(* Logix 5000 project; controller ODSI_Testing vendor 1 type 14 code 151 rev 20.19; software revision 20.05 *)

TASK MainTask (continuous, watchdog 500 ms) : MainProgram

MODULES
   Local : vendor 1 type 14 code 151 (Compact 0, rev 20.19)
      ExpansionInput : 1769-IQ16 (Compact 4, rev 1.1, Input RPI 20 ms)   // Sink or Source
      Discrete_IO : Embedded (Compact 1, rev 3.1, Output RPI 20 ms)
      Analog_IO : Embedded (Compact 2, rev 1.1, Output RPI 80 ms)
      Counters : Embedded (Compact 3, rev 1.1, Output RPI 20 ms)
END_MODULES

VAR_GLOBAL   (* controller tags *)
   DutyCycleOutput : BOOL := 1;   // 1.25 second duty cycle output
   DutyCycleTimer : TIMER := (PRE := 2500, ACC := 2111, EN := 1, TT := 1);   // Accumulates preset time then resets
   HMI_Stop_R1 : BOOL;   // Stop PB on HMI
   HMI_Stop_R2 : BOOL;   // Stop PB on HMI
   ODSI_Fail_Sample1_R1 : ALIAS FOR Local:4:I.Data.4;   // ODSI sent a fail signal for sample 1
   ODSI_Fail_Sample1_R2 : ALIAS FOR Local:1:I.Data.4;   // ODSI sent a fail signal for sample 1
   ODSI_Fail_Sample2_R1 : ALIAS FOR Local:4:I.Data.6;   // ODSI sent a fail signal for sample 2
   ODSI_Fail_Sample2_R2 : ALIAS FOR Local:1:I.Data.6;   // ODSI sent a fail signal for sample 2
   ODSI_Fail_Sample3_R1 : ALIAS FOR Local:4:I.Data.8;   // ODSI sent a fail signal for sample 3
   ODSI_Fail_Sample3_R2 : ALIAS FOR Local:1:I.Data.8;   // ODSI sent a fail signal for sample 3
   ODSI_Pass_Sample1_R1 : ALIAS FOR Local:4:I.Data.3;   // ODSI sent a pass signal for sample 1
   ODSI_Pass_Sample1_R2 : ALIAS FOR Local:1:I.Data.3;   // ODSI sent a pass signal for sample 1
   ODSI_Pass_Sample2_R1 : ALIAS FOR Local:4:I.Data.5;   // ODSI sent a pass signal for sample 2
   ODSI_Pass_Sample2_R2 : ALIAS FOR Local:1:I.Data.5;   // ODSI sent a pass signal for sample 2
   ODSI_Pass_Sample3_R1 : ALIAS FOR Local:4:I.Data.7;   // ODSI sent a pass signal for sample 3
   ODSI_Pass_Sample3_R2 : ALIAS FOR Local:1:I.Data.7;   // ODSI sent a pass signal for sample 3
   ODSI_Valve1_R1 : ALIAS FOR Local:4:I.Data.0;   // ODSI requests to open valve 1
   ODSI_Valve1_R2 : ALIAS FOR Local:1:I.Data.0;   // ODSI requests to open valve 1
   ODSI_Valve2_R1 : ALIAS FOR Local:4:I.Data.1;   // ODSI requests to open valve 2
   ODSI_Valve2_R2 : ALIAS FOR Local:1:I.Data.1;   // ODSI requests to open valve 2
   ODSI_Valve3_R1 : ALIAS FOR Local:4:I.Data.2;   // ODSI requests to open valve 3
   ODSI_Valve3_R2 : ALIAS FOR Local:1:I.Data.2;   // ODSI requests to open valve 3
   R1_DELAY_ONS : BOOL;
   R2_DELAY_ONS : BOOL;
   RandomDelay : DINT := 11;   // Random number generator 0-19
   RandomDelayDisplay_R1 : DINT;   // Snapshot of random delay at time of valve position request for remote 1
   RandomDelayDisplay_R2 : DINT;   // Snapshot of random delay at time of valve position request for remote 2
   RNG_Delay_Active_R1 : BOOL;   // HMI PB randomizing valve open delay
   RNG_Delay_Active_R2 : BOOL;   // HMI PB randomizing valve open delay
   S1_PB_Input_R1 : BOOL;   // HMI PB requesting sample 1
   S1_PB_Input_R2 : BOOL;   // HMI PB requesting sample 1
   S1_Request_R1 : ALIAS FOR Local:1:O.Data.8;   // Output to ODSI to request Sample 1
   S1_Request_R2 : ALIAS FOR Local:1:O.Data.0;   // Output to ODSI to request Sample 1
   S2_PB_Input_R1 : BOOL;   // HMI PB requesting sample 2
   S2_PB_Input_R2 : BOOL;   // HMI PB requesting sample 2
   S2_Request_R1 : ALIAS FOR Local:1:O.Data.9;   // Output to ODSI to request Sample 2
   S2_Request_R2 : ALIAS FOR Local:1:O.Data.1;   // Output to ODSI to request Sample 2
   S3_PB_Input_R1 : BOOL;   // HMI PB requesting sample 3
   S3_PB_Input_R2 : BOOL;   // HMI PB requesting sample 3
   S3_Request_R1 : ALIAS FOR Local:1:O.Data.10;   // Output to ODSI to request Sample 3
   S3_Request_R2 : ALIAS FOR Local:1:O.Data.2;   // Output to ODSI to request Sample 3
   System_Running_Display_R1 : BOOL;   // Displays system running on HMI
   System_Running_Display_R2 : BOOL;   // Displays system running on HMI
   System_Running_R1 : ALIAS FOR Local:4:I.Data.9;   // ODSI signal that indicates the system is currently analyzing a sample
   System_Running_R2 : ALIAS FOR Local:1:I.Data.9;   // ODSI signal that indicates the system is currently analyzing a sample
   SystemTime : DINT[7] := ([0] := 1998, [1] := 1, [2] := 22, [3] := 5, [4] := 42, [5] := 32, [6] := 563285);
        [1]   // Month
        [4]   // Minute
        [0]   // Year
        [2]   // Day
        [3]   // Hour
        [5]   // Second
        [6]   // Microsecond
   Temp : DINT := 10;
   Valve1_Open_Delay_R1 : TIMER;   // Delay after Request is Initiated from ODSI
   Valve1_Open_Delay_R2 : TIMER;   // Delay after Request is Initiated from ODSI
   Valve1_Open_R1 : ALIAS FOR Local:1:O.Data.11;   // Output to ODSI confirming valve 1 is open
   Valve1_Open_R2 : ALIAS FOR Local:1:O.Data.3;   // Output to ODSI confirming valve 1 is open
   Valve1_Open_Random_Delay_R1 : TIMER := (PRE := 11000);   // Randomized delay after request for valve position is received from ODSI
   Valve1_Open_Random_Delay_R2 : TIMER := (PRE := 11000);   // Randomized delay after request for valve position is received from ODSI
   Valve2_Open_Delay_R1 : TIMER;   // Delay after Request is Initiated from ODSI
   Valve2_Open_Delay_R2 : TIMER;   // Delay after Request is Initiated from ODSI
   Valve2_Open_R1 : ALIAS FOR Local:1:O.Data.12;   // Output to ODSI confirming valve 2 is open
   Valve2_Open_R2 : ALIAS FOR Local:1:O.Data.4;   // Output to ODSI confirming valve 2 is open
   Valve2_Open_Random_Delay_R1 : TIMER := (PRE := 11000);   // Randomized delay after request for valve position is received from ODSI
   Valve2_Open_Random_Delay_R2 : TIMER := (PRE := 11000);   // Randomized delay after request for valve position is received from ODSI
   Valve3_Open_Delay_R1 : TIMER;   // Delay after Request is Initiated from ODSI
   Valve3_Open_Delay_R2 : TIMER;   // Delay after Request is Initiated from ODSI
   Valve3_Open_R1 : ALIAS FOR Local:1:O.Data.13;   // Output to ODSI confirming valve 3 is open
   Valve3_Open_R2 : ALIAS FOR Local:1:O.Data.5;   // Output to ODSI confirming valve 3 is open
   Valve3_Open_Random_Delay_R1 : TIMER := (PRE := 11000);   // Randomized delay after request for valve position is received from ODSI
   Valve3_Open_Random_Delay_R2 : TIMER := (PRE := 11000);   // Randomized delay after request for valve position is received from ODSI
   Valve_Block_R1 : BOOL;   // HMI PB to prevent valves from opening
   Valve_Block_R2 : BOOL;   // HMI PB to prevent valves from opening
   Valve_Delay_R1 : DINT;
   Valve_Delay_R2 : DINT;
   Valve_Open_Delay_R2 : TIMER := (PRE := 10000);   // Delay after Request is Initiated from ODSI
END_VAR

PROGRAM MainProgram   (* main routine MainRoutine *)

ROUTINE MainRoutine   (* ladder *)
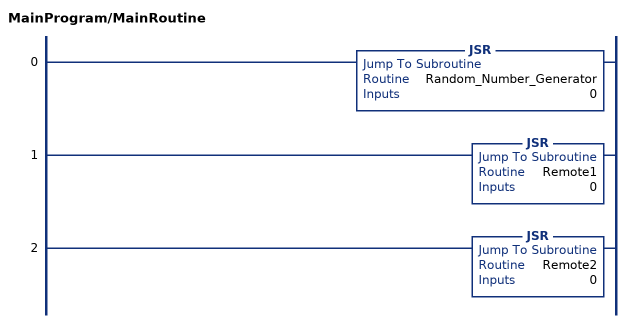
   0: JSR(Random_Number_Generator,0);
   1: JSR(Remote1,0);
   2: JSR(Remote2,0);
END_ROUTINE

ROUTINE Random_Number_Generator   (* ladder *)
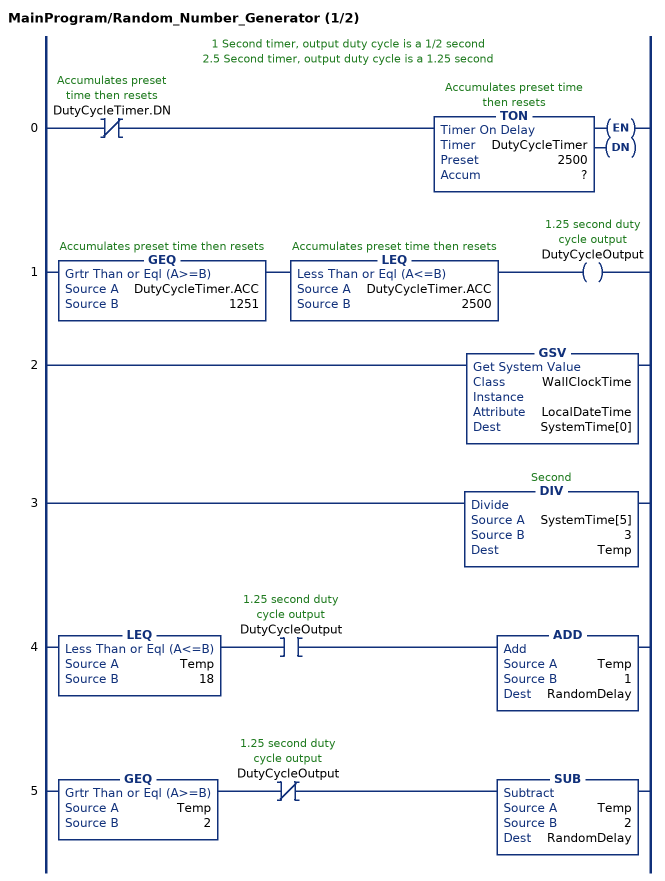
   // 1 Second timer, output duty cycle is a 1/2 second
   // 2.5 Second timer, output duty cycle is a 1.25 second
   0: XIO(DutyCycleTimer.DN)TON(DutyCycleTimer,?,?);
   1: GEQ(DutyCycleTimer.ACC,1251)LEQ(DutyCycleTimer.ACC,2500)OTE(DutyCycleOutput);
   2: GSV(WallClockTime,,LocalDateTime,SystemTime[0]);
   3: DIV(SystemTime[5],3,Temp);
   4: LEQ(Temp,18)XIC(DutyCycleOutput)ADD(Temp,1,RandomDelay);
   5: GEQ(Temp,2)XIO(DutyCycleOutput)SUB(Temp,2,RandomDelay);
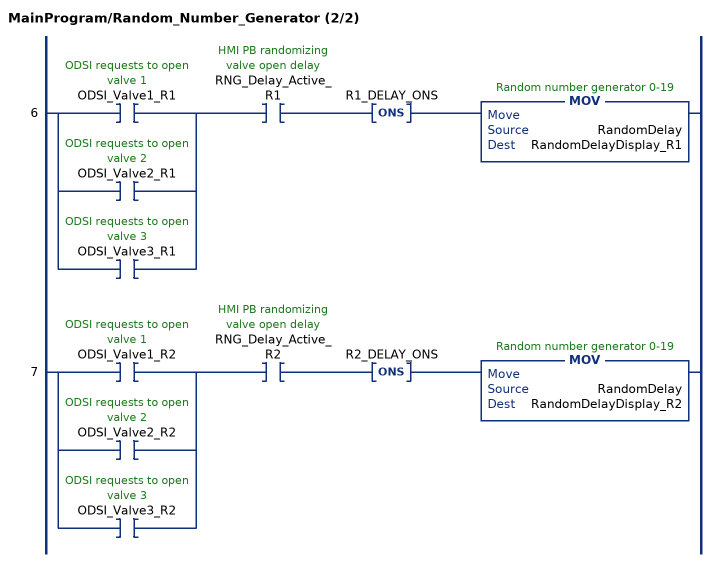
   6: [XIC(ODSI_Valve1_R1) ,XIC(ODSI_Valve2_R1) ,XIC(ODSI_Valve3_R1) ]XIC(RNG_Delay_Active_R1)ONS(R1_DELAY_ONS)MOV(RandomDelay,RandomDelayDisplay_R1);
   7: [XIC(ODSI_Valve1_R2) ,XIC(ODSI_Valve2_R2) ,XIC(ODSI_Valve3_R2) ]XIC(RNG_Delay_Active_R2)ONS(R2_DELAY_ONS)MOV(RandomDelay,RandomDelayDisplay_R2);
END_ROUTINE

ROUTINE Remote1   (* ladder *)
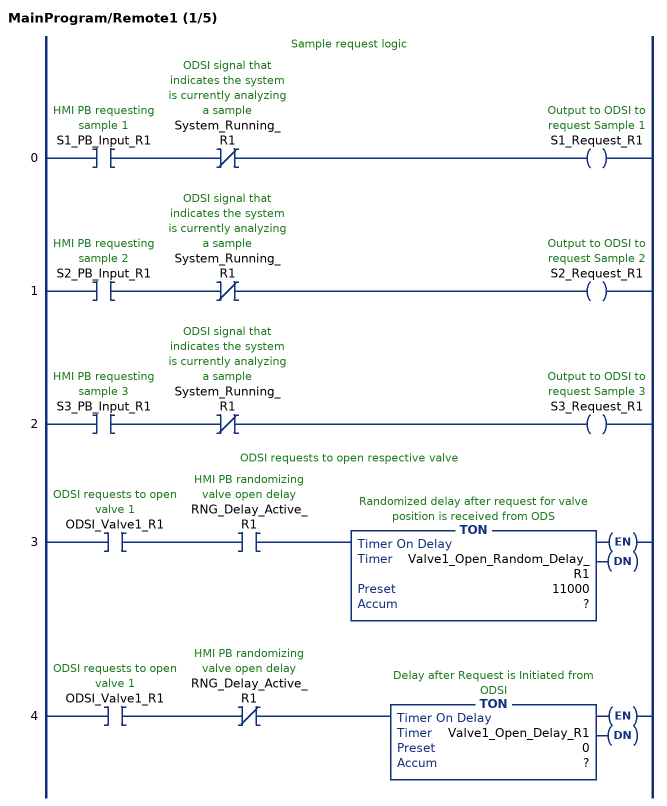
   // Sample request logic
   0: XIC(S1_PB_Input_R1)XIO(System_Running_R1)OTE(S1_Request_R1);
   1: XIC(S2_PB_Input_R1)XIO(System_Running_R1)OTE(S2_Request_R1);
   2: XIC(S3_PB_Input_R1)XIO(System_Running_R1)OTE(S3_Request_R1);
   // ODSI requests to open respective valve
   3: XIC(ODSI_Valve1_R1)XIC(RNG_Delay_Active_R1)TON(Valve1_Open_Random_Delay_R1,?,?);
   4: XIC(ODSI_Valve1_R1)XIO(RNG_Delay_Active_R1)TON(Valve1_Open_Delay_R1,?,?);
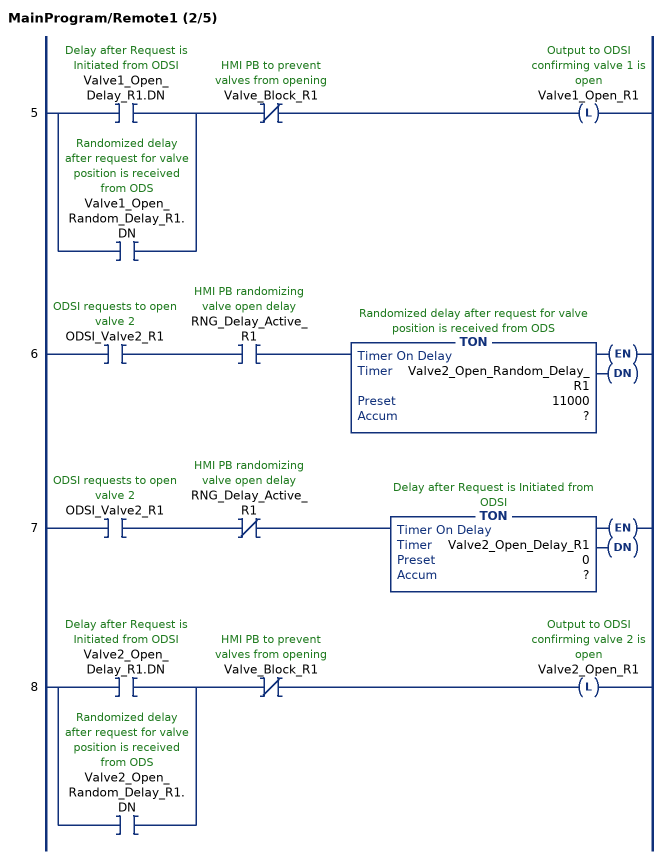
   5: [XIC(Valve1_Open_Delay_R1.DN) ,XIC(Valve1_Open_Random_Delay_R1.DN) ]XIO(Valve_Block_R1)OTL(Valve1_Open_R1);
   6: XIC(ODSI_Valve2_R1)XIC(RNG_Delay_Active_R1)TON(Valve2_Open_Random_Delay_R1,?,?);
   7: XIC(ODSI_Valve2_R1)XIO(RNG_Delay_Active_R1)TON(Valve2_Open_Delay_R1,?,?);
   8: [XIC(Valve2_Open_Delay_R1.DN) ,XIC(Valve2_Open_Random_Delay_R1.DN) ]XIO(Valve_Block_R1)OTL(Valve2_Open_R1);
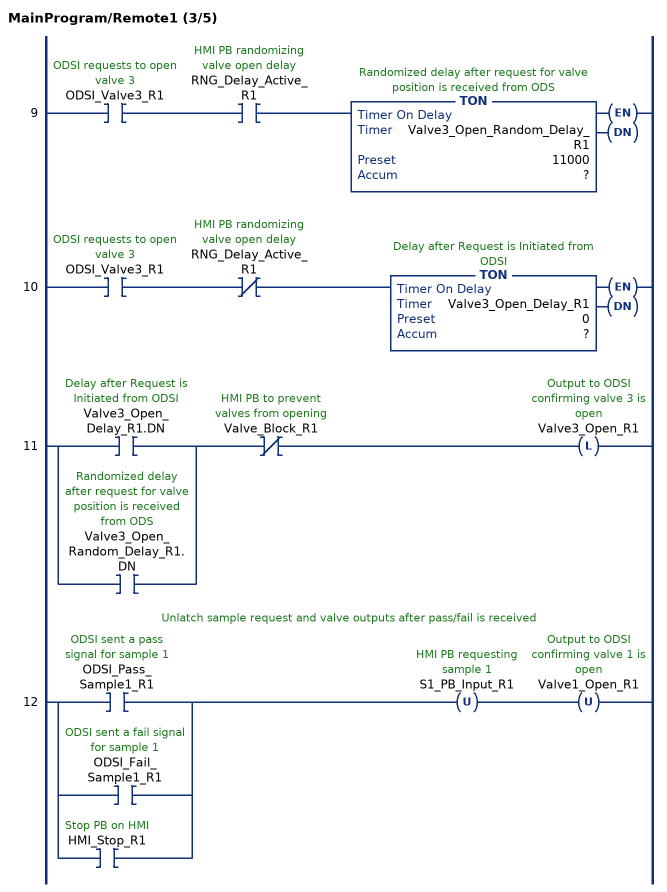
   9: XIC(ODSI_Valve3_R1)XIC(RNG_Delay_Active_R1)TON(Valve3_Open_Random_Delay_R1,?,?);
   10: XIC(ODSI_Valve3_R1)XIO(RNG_Delay_Active_R1)TON(Valve3_Open_Delay_R1,?,?);
   11: [XIC(Valve3_Open_Delay_R1.DN) ,XIC(Valve3_Open_Random_Delay_R1.DN) ]XIO(Valve_Block_R1)OTL(Valve3_Open_R1);
   // Unlatch sample request and valve outputs after pass/fail is received
   12: [XIC(ODSI_Pass_Sample1_R1) ,XIC(ODSI_Fail_Sample1_R1) ,XIC(HMI_Stop_R1) ]OTU(S1_PB_Input_R1)OTU(Valve1_Open_R1);
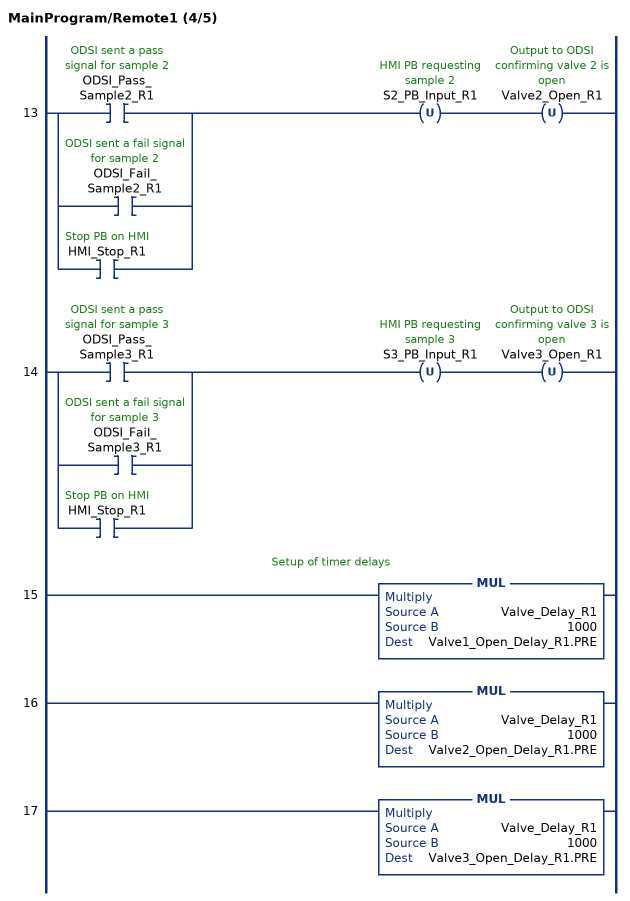
   13: [XIC(ODSI_Pass_Sample2_R1) ,XIC(ODSI_Fail_Sample2_R1) ,XIC(HMI_Stop_R1) ]OTU(S2_PB_Input_R1)OTU(Valve2_Open_R1);
   14: [XIC(ODSI_Pass_Sample3_R1) ,XIC(ODSI_Fail_Sample3_R1) ,XIC(HMI_Stop_R1) ]OTU(S3_PB_Input_R1)OTU(Valve3_Open_R1);
   // Setup of timer delays
   15: MUL(Valve_Delay_R1,1000,Valve1_Open_Delay_R1.PRE);
   16: MUL(Valve_Delay_R1,1000,Valve2_Open_Delay_R1.PRE);
   17: MUL(Valve_Delay_R1,1000,Valve3_Open_Delay_R1.PRE);
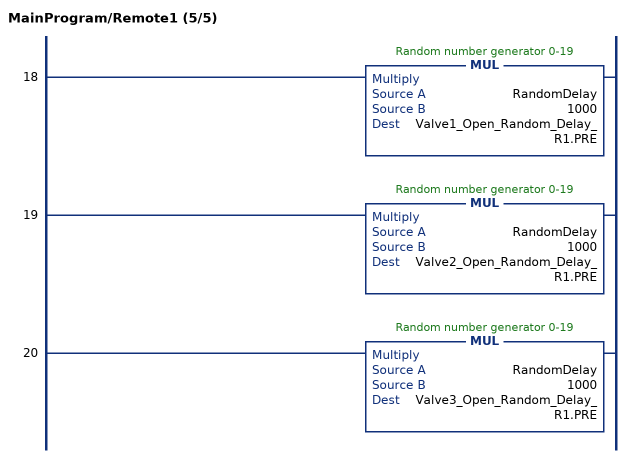
   18: MUL(RandomDelay,1000,Valve1_Open_Random_Delay_R1.PRE);
   19: MUL(RandomDelay,1000,Valve2_Open_Random_Delay_R1.PRE);
   20: MUL(RandomDelay,1000,Valve3_Open_Random_Delay_R1.PRE);
END_ROUTINE

ROUTINE Remote2   (* ladder *)
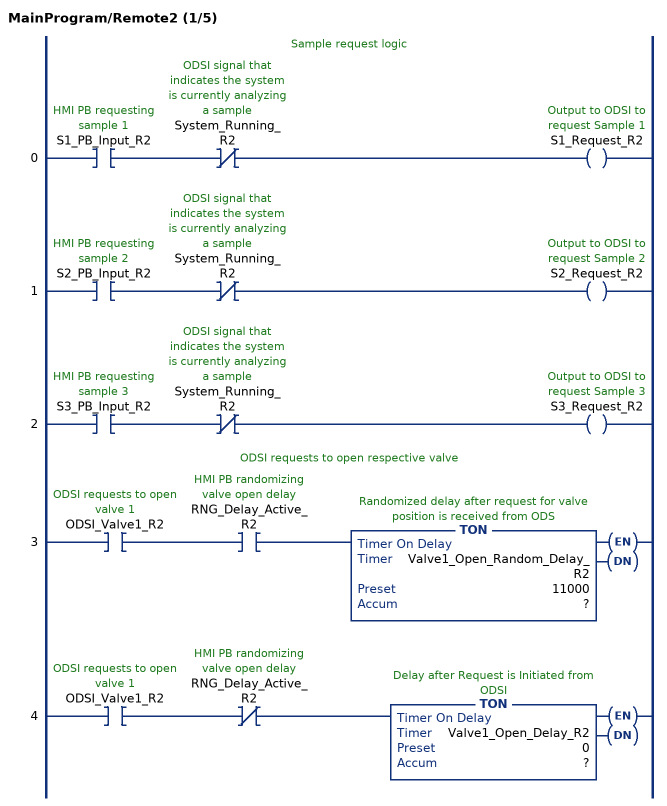
   // Sample request logic
   0: XIC(S1_PB_Input_R2)XIO(System_Running_R2)OTE(S1_Request_R2);
   1: XIC(S2_PB_Input_R2)XIO(System_Running_R2)OTE(S2_Request_R2);
   2: XIC(S3_PB_Input_R2)XIO(System_Running_R2)OTE(S3_Request_R2);
   // ODSI requests to open respective valve
   3: XIC(ODSI_Valve1_R2)XIC(RNG_Delay_Active_R2)TON(Valve1_Open_Random_Delay_R2,?,?);
   4: XIC(ODSI_Valve1_R2)XIO(RNG_Delay_Active_R2)TON(Valve1_Open_Delay_R2,?,?);
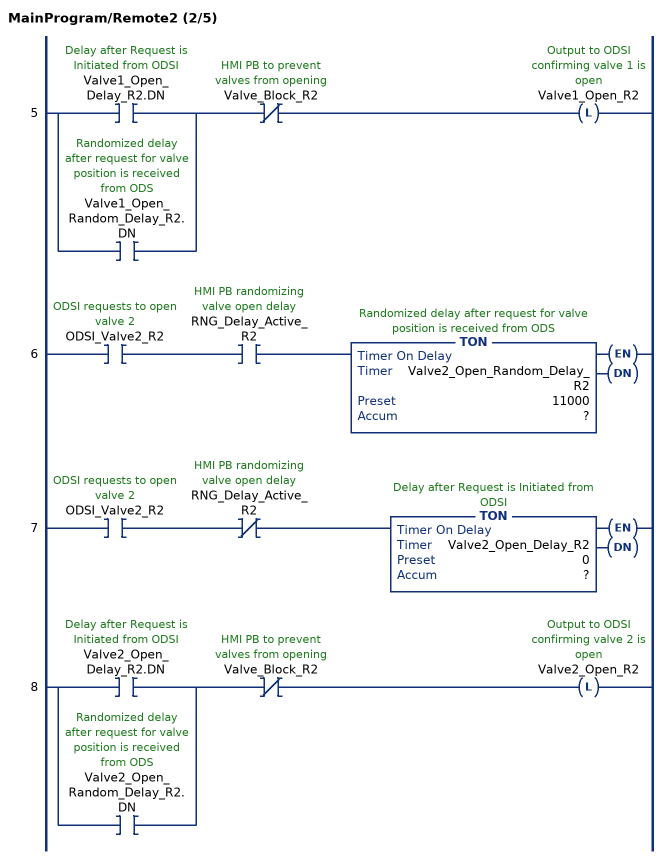
   5: [XIC(Valve1_Open_Delay_R2.DN) ,XIC(Valve1_Open_Random_Delay_R2.DN) ]XIO(Valve_Block_R2)OTL(Valve1_Open_R2);
   6: XIC(ODSI_Valve2_R2)XIC(RNG_Delay_Active_R2)TON(Valve2_Open_Random_Delay_R2,?,?);
   7: XIC(ODSI_Valve2_R2)XIO(RNG_Delay_Active_R2)TON(Valve2_Open_Delay_R2,?,?);
   8: [XIC(Valve2_Open_Delay_R2.DN) ,XIC(Valve2_Open_Random_Delay_R2.DN) ]XIO(Valve_Block_R2)OTL(Valve2_Open_R2);
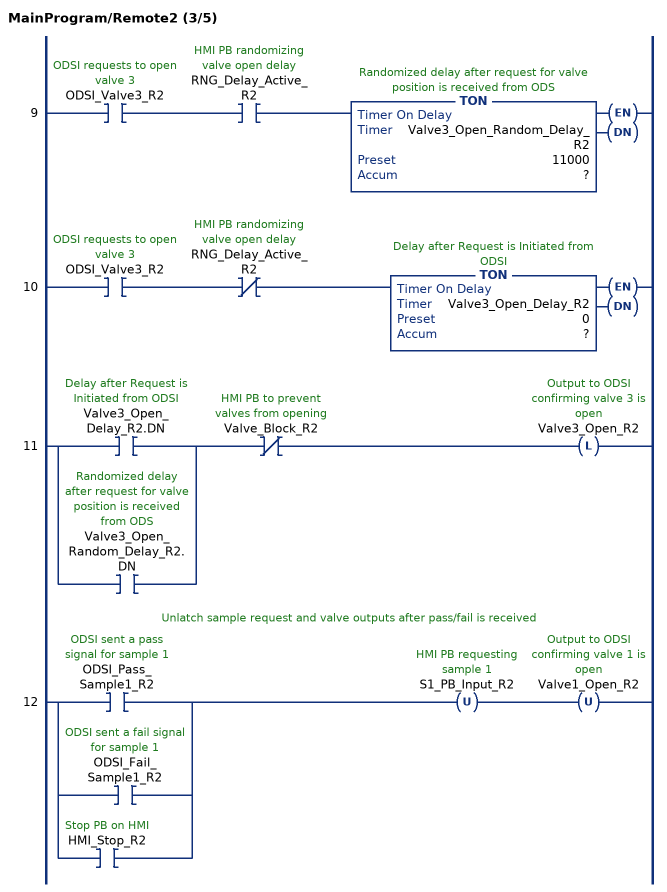
   9: XIC(ODSI_Valve3_R2)XIC(RNG_Delay_Active_R2)TON(Valve3_Open_Random_Delay_R2,?,?);
   10: XIC(ODSI_Valve3_R2)XIO(RNG_Delay_Active_R2)TON(Valve3_Open_Delay_R2,?,?);
   11: [XIC(Valve3_Open_Delay_R2.DN) ,XIC(Valve3_Open_Random_Delay_R2.DN) ]XIO(Valve_Block_R2)OTL(Valve3_Open_R2);
   // Unlatch sample request and valve outputs after pass/fail is received
   12: [XIC(ODSI_Pass_Sample1_R2) ,XIC(ODSI_Fail_Sample1_R2) ,XIC(HMI_Stop_R2) ]OTU(S1_PB_Input_R2)OTU(Valve1_Open_R2);
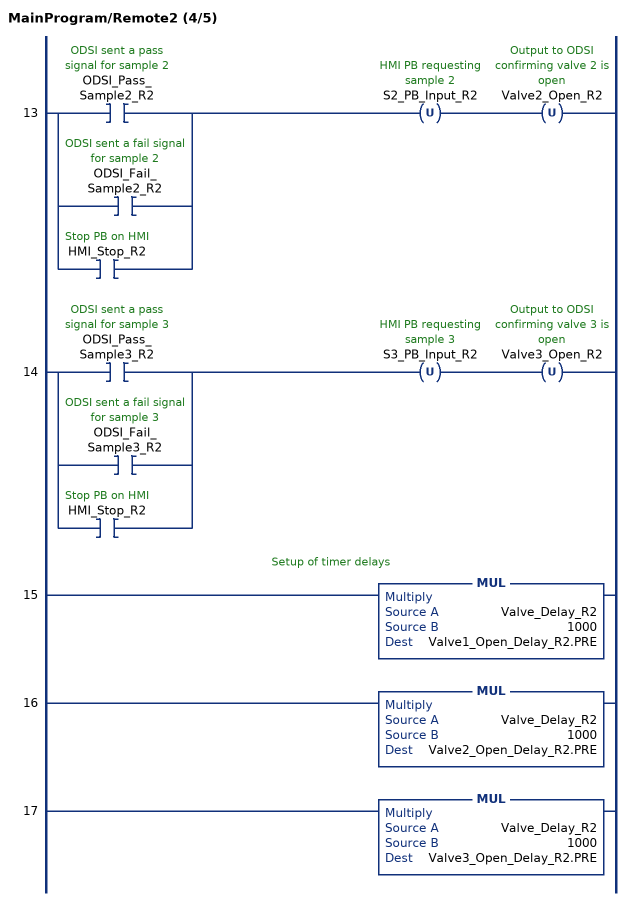
   13: [XIC(ODSI_Pass_Sample2_R2) ,XIC(ODSI_Fail_Sample2_R2) ,XIC(HMI_Stop_R2) ]OTU(S2_PB_Input_R2)OTU(Valve2_Open_R2);
   14: [XIC(ODSI_Pass_Sample3_R2) ,XIC(ODSI_Fail_Sample3_R2) ,XIC(HMI_Stop_R2) ]OTU(S3_PB_Input_R2)OTU(Valve3_Open_R2);
   // Setup of timer delays
   15: MUL(Valve_Delay_R2,1000,Valve1_Open_Delay_R2.PRE);
   16: MUL(Valve_Delay_R2,1000,Valve2_Open_Delay_R2.PRE);
   17: MUL(Valve_Delay_R2,1000,Valve3_Open_Delay_R2.PRE);
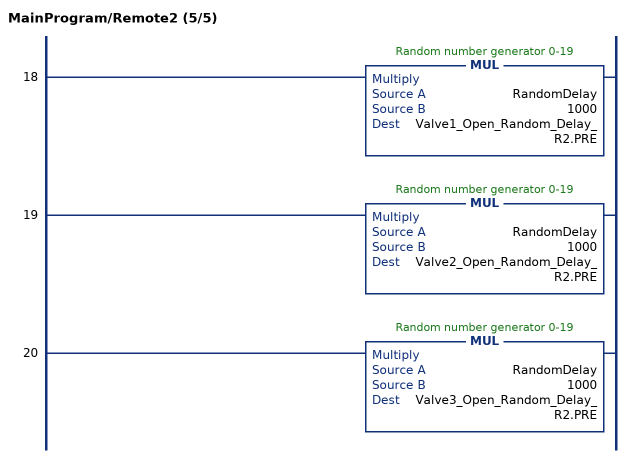
   18: MUL(RandomDelay,1000,Valve1_Open_Random_Delay_R2.PRE);
   19: MUL(RandomDelay,1000,Valve2_Open_Random_Delay_R2.PRE);
   20: MUL(RandomDelay,1000,Valve3_Open_Random_Delay_R2.PRE);
END_ROUTINE
END_PROGRAM
